(*********************************** G.D S.p.A. - Technical Department ***********************************
============= PROGRAM INFO ============
FOLDER:             TBD
MACHINES INVOLVED:  TBD 

============= DESCRIPTION =============

============= REVISIONS ===============
Date		Version	 	Author      	Description             
----------	-------		------------  	--------------------------------------------
2019/10/07 	0000.00	 	W.Gerstner		Creation of the PRG

**********************************************************************************************************)
(*$R
	process_ref := prc;
$*)
PROGRAM csp_case_main_services_vacuum
VAR
	prc:					process;
	prc_path:				STRING;
END_VAR

_read_var_input();

_object_manager();

IF NOT objects_running()
THEN
	RETURN;	
END_IF

_read_process_image();

_mode_manager();

CASE process_get_mode(prc) of
	MODE_ABSENT,
	MODE_INACTIVE:
		RETURN;
	MODE_TEST:
		_handle_process_test();
END_CASE

_set_runtime_properties();

(********************************* BODY *********************************)

(************************************************************************)

_handle_messages();

_write_output();

ACTION _handle_messages:
;
END_ACTION

ACTION _handle_process_test:
;
END_ACTION

ACTION _mode_manager:
IF process_mode_req_is_pending(prc)
THEN
    process_apply_mode_req_first_step(prc);
    CASE process_get_mode(prc) OF
        MODE_TO_ABSENT:
			;
        MODE_TO_INACTIVE:
			;
        MODE_TO_TEST:
			;
        MODE_TO_OPERATIONAL:
			;
    END_CASE
    process_apply_mode_req_second_step(prc);
END_IF
END_ACTION

ACTION _object_manager:
IF objects_initialization()
THEN
	sub_process_init(
		object_name						:= 'csp_case_main_services_vacuum.prc', 
		process							:= csp_case_main_services.prc, 
		CONVERSION_this					:= prc);
		
	prc_path 							:= process_get_path(prc);
END_IF

IF objects_running()
THEN
	process_cycle(prc);
END_IF
END_ACTION

ACTION _read_process_image:
;
END_ACTION

ACTION _read_var_input:
;
END_ACTION

ACTION _set_runtime_properties:
;
END_ACTION

ACTION _write_output:
;
END_ACTION

END_PROGRAM

(* stored: Version 1.1.0.1, ProductVersion 3.1.4022.12
   POU csp_case_main_services_vacuum: Id {5c460230-ee4e-479c-87a0-44aca56e542c}, SpecialFunc None
   Action _handle_messages: Id {51c5d9fe-cc48-49fc-82ed-ce5b94bd0b98}
   Action _handle_process_test: Id {d24e5538-37c6-45de-a2dd-8f2eb01668e1}
   Action _mode_manager: Id {1058d1c0-66dc-470d-a718-7fa506ed503c}
   Action _object_manager: Id {b9ccbbab-8b2c-4d71-a692-782f7e9b287d}
   Action _read_process_image: Id {93eb9797-94a3-4aa0-9060-78086e4cc478}
   Action _read_var_input: Id {23122c11-2791-4a71-b008-7975cc06b2c2}
   Action _set_runtime_properties: Id {7a415af4-3dd9-42b2-9a6e-c69c2d4a219c}
   Action _write_output: Id {1c2bc031-78a9-4828-a2ed-7c3f3d233196} *)
